// TIA Portal V20 export
FUNCTION_BLOCK "05 T5 EXCENTRIC Sequence"   // FB1518, GRAPH
// stored: AutoNumber false, GraphVersion 6.0, InitialValuesAcquisition false, SetENOAutomatically false
   // inherited from GRAPH_BASE
   VAR_INPUT
      OFF_SQ : Bool := false;
      INIT_SQ : Bool := false;
      ACK_EF : Bool := false;
      S_PREV : Bool := false;
      S_NEXT : Bool := false;
      SW_AUTO : Bool := false;
      SW_TAP : Bool := false;
      SW_TOP : Bool := false;
      SW_MAN : Bool := false;
      S_SEL : Int := 0;
      S_ON : Bool := false;
      S_OFF : Bool := false;
      T_PUSH : Bool := false;
   END_VAR
   VAR_OUTPUT
      S_NO : Int := 0;
      S_MORE : Bool := false;
      S_ACTIVE : Bool := false;
      ERR_FLT : Bool := false;
      AUTO_ON : Bool := false;
      TAP_ON : Bool := false;
      TOP_ON : Bool := false;
      MAN_ON : Bool := false;
   END_VAR
BEGIN
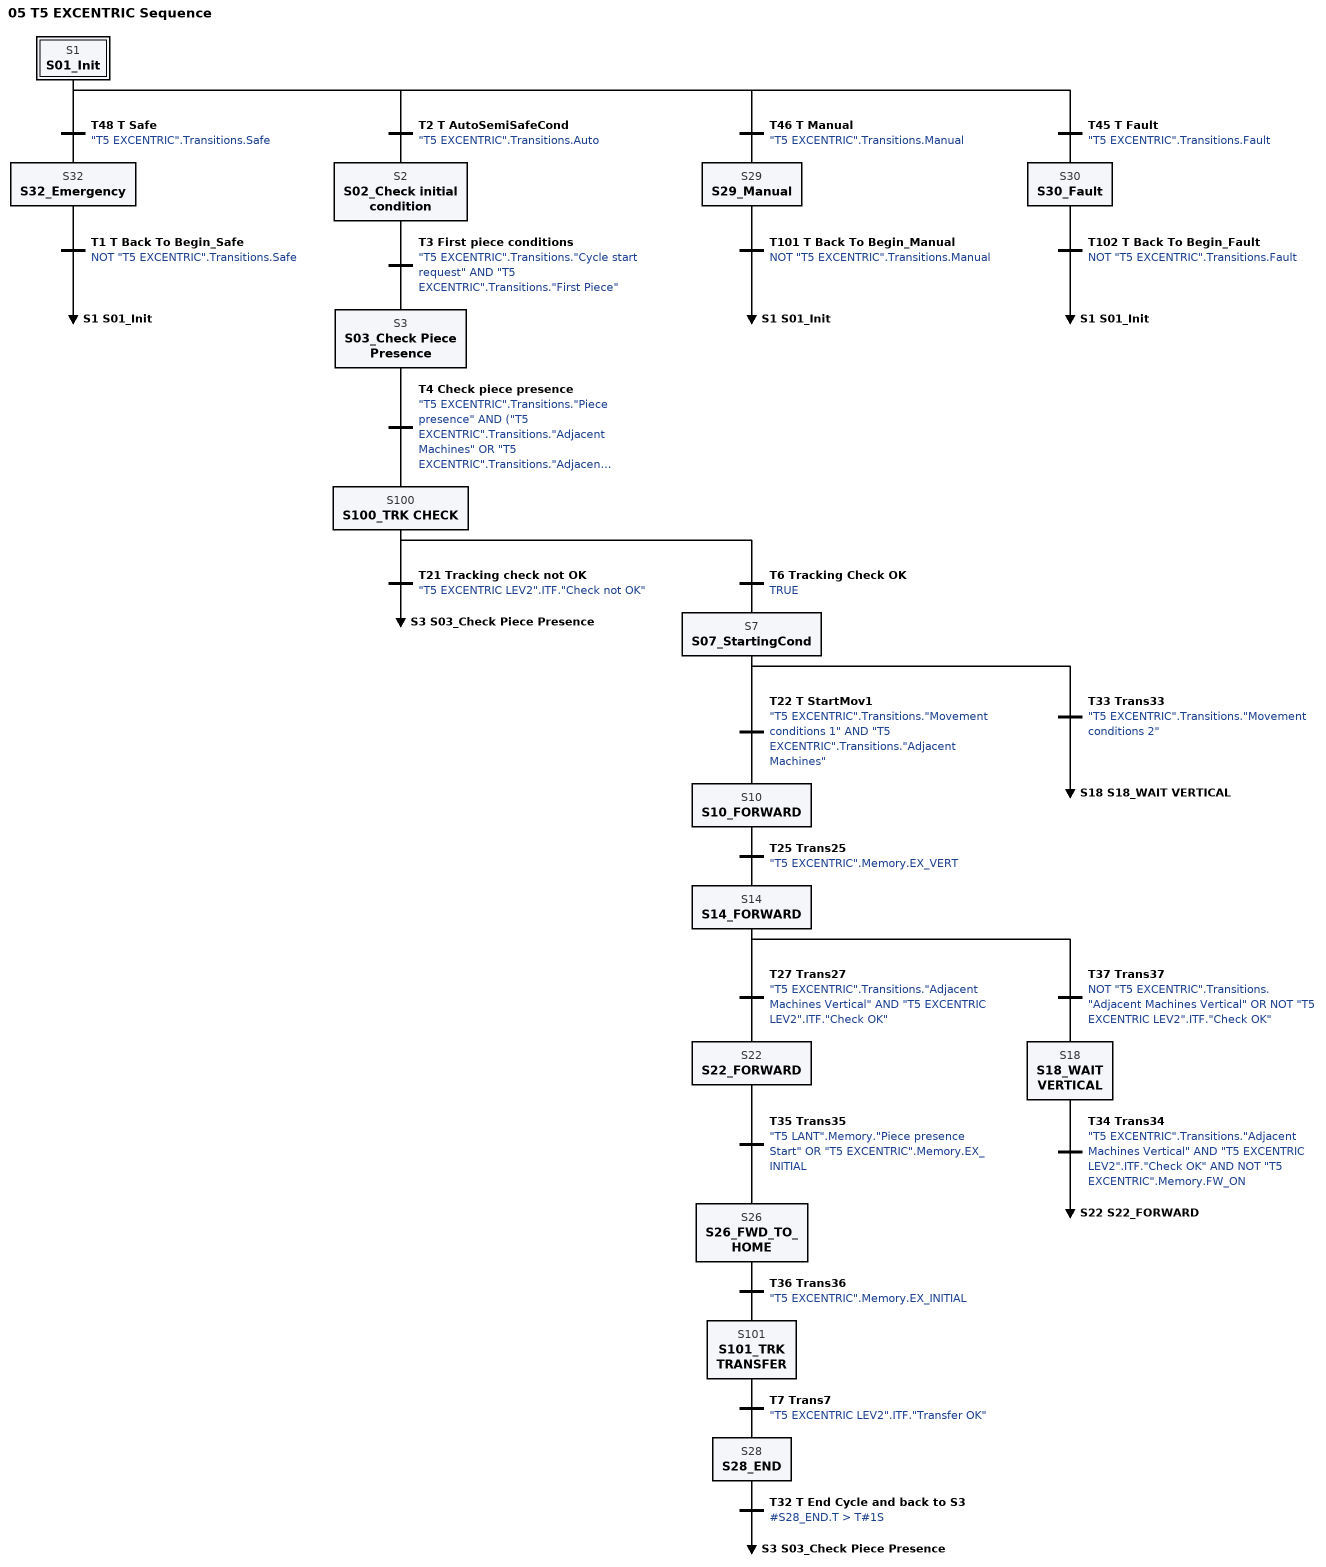
   // permanent pre-instructions
   NETWORK 1
      "01 T5 EXCENTRIC Alarms"();
   NETWORK 2
      "02 T5 EXCENTRIC HMI"();
   NETWORK 3
      "03 T5 EXCENTRIC Aux"();
   NETWORK 4
      "04 T5 EXCENTRIC Transitions"();

   // sequencer 1
   INITIAL_STEP S01_Init:   // S1, max time T#10S, warning time T#7S
   END_STEP
   TRANSITION "T Safe" FROM S01_Init TO S32_Emergency   // T48
      := "T5 EXCENTRIC".Transitions.Safe;
   END_TRANSITION
   TRANSITION "T AutoSemiSafeCond" FROM S01_Init TO "S02_Check initial condition"   // T2
      := "T5 EXCENTRIC".Transitions.Auto;
   END_TRANSITION
   TRANSITION "T Manual" FROM S01_Init TO S29_Manual   // T46
      := "T5 EXCENTRIC".Transitions.Manual;
   END_TRANSITION
   TRANSITION "T Fault" FROM S01_Init TO S30_Fault   // T45
      := "T5 EXCENTRIC".Transitions.Fault;
   END_TRANSITION
   STEP "S03_Check Piece Presence":   // S3, max time T#10S, warning time T#7S
   END_STEP
   TRANSITION "Check piece presence" FROM "S03_Check Piece Presence" TO "S100_TRK CHECK"   // T4
      := "T5 EXCENTRIC".Transitions."Piece presence" AND ("T5 EXCENTRIC".Transitions."Adjacent Machines" OR "T5 EXCENTRIC".Transitions."Adjacent Machines Vertical") AND NOT "T5 EXCENTRIC".Transitions.Pause;
   END_TRANSITION
   STEP S32_Emergency:   // S32, max time T#10S, warning time T#7S
   END_STEP
   TRANSITION "T Back To Begin_Safe" FROM S32_Emergency TO S01_Init   // T1, jump
      := NOT "T5 EXCENTRIC".Transitions.Safe;
   END_TRANSITION
   STEP S29_Manual:   // S29, max time T#10S, warning time T#7S
   END_STEP
   TRANSITION "T Back To Begin_Manual" FROM S29_Manual TO S01_Init   // T101, jump
      := NOT "T5 EXCENTRIC".Transitions.Manual;
   END_TRANSITION
   STEP "S02_Check initial condition":   // S2, max time T#10S, warning time T#7S
   END_STEP
   TRANSITION "First piece conditions" FROM "S02_Check initial condition" TO "S03_Check Piece Presence"   // T3
      := "T5 EXCENTRIC".Transitions."Cycle start request" AND "T5 EXCENTRIC".Transitions."First Piece";
   END_TRANSITION
   STEP S30_Fault:   // S30, max time T#10S, warning time T#7S
   END_STEP
   TRANSITION "T Back To Begin_Fault" FROM S30_Fault TO S01_Init   // T102, jump
      := NOT "T5 EXCENTRIC".Transitions.Fault;
   END_TRANSITION
   STEP S28_END:   // S28, max time T#10S, warning time T#7S
   END_STEP
   TRANSITION "T End Cycle and back to S3" FROM S28_END TO "S03_Check Piece Presence"   // T32, jump: Assenza pezzo o ok da robot
      := #S28_END.T > T#1S;
   END_TRANSITION
   STEP S10_FORWARD:   // S10, max time T#10S, warning time T#7S
   END_STEP
   TRANSITION Trans25 FROM S10_FORWARD TO S14_FORWARD   // T25
      := "T5 EXCENTRIC".Memory.EX_VERT;
   END_TRANSITION
   STEP S14_FORWARD:   // S14, max time T#10S, warning time T#7S
   END_STEP
   TRANSITION Trans27 FROM S14_FORWARD TO S22_FORWARD   // T27
      := "T5 EXCENTRIC".Transitions."Adjacent Machines Vertical" AND "T5 EXCENTRIC LEV2".ITF."Check OK";
   END_TRANSITION
   TRANSITION Trans37 FROM S14_FORWARD TO "S18_WAIT VERTICAL"   // T37
      := NOT "T5 EXCENTRIC".Transitions."Adjacent Machines Vertical" OR NOT "T5 EXCENTRIC LEV2".ITF."Check OK";
   END_TRANSITION
   STEP S22_FORWARD:   // S22, max time T#10S, warning time T#7S
   END_STEP
   TRANSITION Trans35 FROM S22_FORWARD TO S26_FWD_TO_HOME   // T35
      := "T5 LANT".Memory."Piece presence Start" OR "T5 EXCENTRIC".Memory.EX_INITIAL;
   END_TRANSITION
   STEP "S100_TRK CHECK":   // S100, max time T#10S, warning time T#7S
   END_STEP
   TRANSITION "Tracking check not OK" FROM "S100_TRK CHECK" TO "S03_Check Piece Presence"   // T21, jump
      := "T5 EXCENTRIC LEV2".ITF."Check not OK";
   END_TRANSITION
   TRANSITION "Tracking Check OK" FROM "S100_TRK CHECK" TO S07_StartingCond   // T6
      := TRUE;
   END_TRANSITION
   STEP "S18_WAIT VERTICAL":   // S18, max time T#10S, warning time T#7S
   END_STEP
   TRANSITION Trans34 FROM "S18_WAIT VERTICAL" TO S22_FORWARD   // T34, jump
      := "T5 EXCENTRIC".Transitions."Adjacent Machines Vertical" AND "T5 EXCENTRIC LEV2".ITF."Check OK" AND NOT "T5 EXCENTRIC".Memory.FW_ON;
   END_TRANSITION
   STEP S07_StartingCond:   // S7, max time T#10S, warning time T#7S
   END_STEP
   TRANSITION "T StartMov1" FROM S07_StartingCond TO S10_FORWARD   // T22
      := "T5 EXCENTRIC".Transitions."Movement conditions 1" AND "T5 EXCENTRIC".Transitions."Adjacent Machines";
   END_TRANSITION
   TRANSITION Trans33 FROM S07_StartingCond TO "S18_WAIT VERTICAL"   // T33, jump
      := "T5 EXCENTRIC".Transitions."Movement conditions 2";
   END_TRANSITION
   STEP S26_FWD_TO_HOME:   // S26, max time T#10S, warning time T#7S
   END_STEP
   TRANSITION Trans36 FROM S26_FWD_TO_HOME TO "S101_TRK TRANSFER"   // T36
      := "T5 EXCENTRIC".Memory.EX_INITIAL;
   END_TRANSITION
   STEP "S101_TRK TRANSFER":   // S101, max time T#10S, warning time T#7S
   END_STEP
   TRANSITION Trans7 FROM "S101_TRK TRANSFER" TO S28_END   // T7
      := "T5 EXCENTRIC LEV2".ITF."Transfer OK";
   END_TRANSITION

   // permanent post-instructions
   NETWORK 1
      "06 T5 EXCENTRIC Output"();
   NETWORK 2
      "07 T5 EXCENTRIC LEV2"();
END_FUNCTION_BLOCK
